{attribute addProperty BoxType "EL2014-0000-0016"}
{attribute addProperty Id "ChannelAT %I*ARRAY[0 ..3] OF Channel_38C6D80F1620"}
{attribute addProperty CRC "3399384941"}
{attribute addProperty SizeInBites "16"}
{attribute addProperty SizeInBytes "2"}
TYPE DIG_Diag_Inputs_B107C8FA :
STRUCT
	{attribute addProperty Name "Channel"}
	Channel AT %I* : ARRAY[0 ..3] OF Channel_38C6D80F;
END_STRUCT
END_TYPE

(* stored: Version 1.2.0.0, ProductVersion 3.1.4024.9
   DUT DIG_Diag_Inputs_B107C8FA: Id {f162df32-3184-461a-a147-87cb12f23cd4} *)
